LIN {X 0,Y 77.995,Z 481.721,A -85,B 0,C 180,E1 -30607.645,E2 -30607.645} C_VEL
LIN {X 0,Y 72.024,Z 491.434,A -85,B 0,C 180,E1 -30608.921,E2 -30608.921} C_VEL
LIN {X 0,Y 64.422,Z 501.593,A -85,B 0,C 180,E1 -30610.964,E2 -30610.964} C_VEL
LIN {X 0,Y 55.946,Z 510.931,A -85,B 0,C 180,E1 -30613.993,E2 -30613.993} C_VEL
LIN {X 0,Y 48.02,Z 518.337,A -85,B 0,C 180,E1 -30617.976,E2 -30617.976} C_VEL
LIN {X 0,Y 38.72,Z 525.749,A -85,B 0,C 180,E1 -30624.852,E2 -30624.852} C_VEL
LIN {X 0,Y 30.186,Z 531.666,A -85,B 0,C 180,E1 -30635.441,E2 -30635.441} C_VEL
LIN {X 0,Y 23.499,Z 536.326,A -85,B 0,C 180,E1 -30653.279,E2 -30653.279} C_VEL
LIN {X 0,Y 20.813,Z 538.779,A -85,B 0,C 180,E1 -30670.28,E2 -30670.28} C_VEL
LIN {X 0,Y 20.096,Z 540.766,A -85,B 0,C 180,E1 -30690.015,E2 -30690.015} C_VEL
LIN {X 0,Y 20.854,Z 542.293,A -85,B 0,C 180,E1 -30709.71,E2 -30709.71} C_VEL
LIN {X 0,Y 23.631,Z 543.406,A -85,B 0,C 180,E1 -30726.514,E2 -30726.514} C_VEL
LIN {X 0,Y 33.09,Z 544.394,A -85,B 0,C 180,E1 -30748.179,E2 -30748.179} C_VEL
LIN {X 0,Y 45.153,Z 543.887,A -85,B 0,C 180,E1 -30759.066,E2 -30759.066} C_VEL
LIN {X 0,Y 51.564,Z 543.027,A -85,B 0,C 180,E1 -30762.585,E2 -30762.585} C_VEL
LIN {X 0,Y 64.818,Z 540.118,A -85,B 0,C 180,E1 -30767.397,E2 -30767.397} C_VEL
LIN {X 0,Y 74.959,Z 536.824,A -85,B 0,C 180,E1 -30769.904,E2 -30769.904} C_VEL
LIN {X 0,Y 85.212,Z 532.49,A -85,B 0,C 180,E1 -30771.796,E2 -30771.796} C_VEL
LIN {X 0,Y 97.293,Z 525.973,A -85,B 0,C 180,E1 -30773.354,E2 -30773.354} C_VEL
LIN {X 0,Y 107.703,Z 518.838,A -85,B 0,C 180,E1 -30774.356,E2 -30774.356} C_VEL
LIN {X 0,Y 112.916,Z 514.651,A -85,B 0,C 180,E1 -30774.804,E2 -30774.804} C_VEL
LIN {X 0,Y 112.809,Z 514.716,A -85,B 0,C 180,E1 -30775.439,E2 -30775.439} C_VEL
LIN {X 0,Y 101.916,Z 522.899,A -85,B 0,C 180,E1 -30776.583,E2 -30776.583} C_VEL
LIN {X 0,Y 91.427,Z 529.167,A -85,B 0,C 180,E1 -30777.944,E2 -30777.944} C_VEL
LIN {X 0,Y 79.346,Z 534.816,A -85,B 0,C 180,E1 -30780.001,E2 -30780.001} C_VEL
LIN {X 0,Y 70.327,Z 538.074,A -85,B 0,C 180,E1 -30781.999,E2 -30781.999} C_VEL
LIN {X 0,Y 63.406,Z 540.049,A -85,B 0,C 180,E1 -30783.942,E2 -30783.942} C_VEL
LIN {X 0,Y 53.983,Z 542.04,A -85,B 0,C 180,E1 -30787.482,E2 -30787.482} C_VEL
LIN {X 0,Y 43.35,Z 543.328,A -85,B 0,C 180,E1 -30793.385,E2 -30793.385} C_VEL
LIN {X 0,Y 37.114,Z 543.588,A -85,B 0,C 180,E1 -30798.746,E2 -30798.746} C_VEL
LIN {X 0,Y 30.404,Z 543.36,A -85,B 0,C 180,E1 -30807.539,E2 -30807.539} C_VEL
LIN {X 0,Y 22.114,Z 541.861,A -85,B 0,C 180,E1 -30830.518,E2 -30830.518} C_VEL
LIN {X 0,Y 19.731,Z 540.267,A -85,B 0,C 180,E1 -30851.546,E2 -30851.546} C_VEL
LIN {X 0,Y 19.099,Z 538.846,A -85,B 0,C 180,E1 -30868.347,E2 -30868.347} C_VEL
LIN {X 0,Y 19.091,Z 537.172,A -85,B 0,C 180,E1 -30885.573,E2 -30885.573} C_VEL
LIN {X 0,Y 22.808,Z 533.113,A -85,B 0,C 180,E1 -30915.29,E2 -30915.29} C_VEL
LIN {X 0,Y 26.639,Z 530.637,A -85,B 0,C 180,E1 -30924.313,E2 -30924.313} C_VEL
LIN {X 0,Y 28.148,Z 529.719,A -85,B 0,C 180,E1 -30926.304,E2 -30926.304} C_VEL
LIN {X 0,Y 38.83,Z 522.853,A -85,B 0,C 180,E1 -30934.8,E2 -30934.8} C_VEL
LIN {X 0,Y 48.8,Z 515.029,A -85,B 0,C 180,E1 -30939.388,E2 -30939.388} C_VEL
LIN {X 0,Y 57.26,Z 507.041,A -85,B 0,C 180,E1 -30942.012,E2 -30942.012} C_VEL
LIN {X 0,Y 65.835,Z 497.276,A -85,B 0,C 180,E1 -30943.88,E2 -30943.88} C_VEL
LIN {X 0,Y 73.637,Z 486.368,A -85,B 0,C 180,E1 -30945.075,E2 -30945.075} C_VEL
LIN {X 0,Y 79.638,Z 475.755,A -85,B 0,C 180,E1 -30946.09,E2 -30946.09} C_VEL
LIN {X 0,Y 85.204,Z 463.02,A -85,B 0,C 180,E1 -30946.976,E2 -30946.976} C_VEL
LIN {X 0,Y 89.274,Z 450.18,A -85,B 0,C 180,E1 -30947.615,E2 -30947.615} C_VEL
LIN {X 0,Y 91.91,Z 437.116,A -85,B 0,C 180,E1 -30948.013,E2 -30948.013} C_VEL
LIN {X 0,Y 92.458,Z 433.099,A -85,B 0,C 180,E1 -30948.178,E2 -30948.178} C_VEL
LIN {X 0,Y 92.246,Z 431.32,A -85,B 0,C 180,E1 -30951.853,E2 -30951.853} C_VEL
LIN {X 0,Y 92.25,Z 430.805,A -85,B 0,C 180,E1 -30955.63,E2 -30955.63} C_VEL
LIN {X 0,Y 92.334,Z 431.487,A -85,B 0,C 180,E1 -30958.091,E2 -30958.091} C_VEL
LIN {X 0,Y 92.506,Z 433,A -85,B 0,C 180,E1 -30960.668,E2 -30960.668} C_VEL
LIN {X 0,Y 90.295,Z 446.232,A -85,B 0,C 180,E1 -30960.99,E2 -30960.99} C_VEL
LIN {X 0,Y 86.533,Z 459.67,A -85,B 0,C 180,E1 -30961.452,E2 -30961.452} C_VEL
LIN {X 0,Y 82.617,Z 469.744,A -85,B 0,C 180,E1 -30961.86,E2 -30961.86} C_VEL
LIN {X 0,Y 76.497,Z 481.913,A -85,B 0,C 180,E1 -30962.508,E2 -30962.508} C_VEL
LIN {X 0,Y 70.397,Z 491.554,A -85,B 0,C 180,E1 -30963.38,E2 -30963.38} C_VEL
LIN {X 0,Y 63.448,Z 500.632,A -85,B 0,C 180,E1 -30964.576,E2 -30964.576} C_VEL
LIN {X 0,Y 54.828,Z 509.947,A -85,B 0,C 180,E1 -30966.645,E2 -30966.645} C_VEL
LIN {X 0,Y 46.073,Z 517.806,A -85,B 0,C 180,E1 -30969.562,E2 -30969.562} C_VEL
LIN {X 0,Y 36.296,Z 525.123,A -85,B 0,C 180,E1 -30974.534,E2 -30974.534} C_VEL
LIN {X 0,Y 26.69,Z 531.123,A -85,B 0,C 180,E1 -30982.866,E2 -30982.866} C_VEL
LIN {X 0,Y 18.291,Z 535.858,A -85,B 0,C 180,E1 -30999.81,E2 -30999.81} C_VEL
LIN {X 0,Y 13.213,Z 539.446,A -85,B 0,C 180,E1 -31034.6,E2 -31034.6} C_VEL
LIN {X 0,Y 12.988,Z 540.398,A -85,B 0,C 180,E1 -31050.023,E2 -31050.023} C_VEL
LIN {X 0,Y 14.361,Z 541.957,A -85,B 0,C 180,E1 -31079.322,E2 -31079.322} C_VEL
LIN {X 0,Y 18.405,Z 543.114,A -85,B 0,C 180,E1 -31099.814,E2 -31099.814} C_VEL
LIN {X 0,Y 23.846,Z 543.844,A -85,B 0,C 180,E1 -31112.174,E2 -31112.174} C_VEL
LIN {X 0,Y 29.951,Z 544.179,A -85,B 0,C 180,E1 -31119.843,E2 -31119.843} C_VEL
LIN {X 0,Y 43.122,Z 543.735,A -85,B 0,C 180,E1 -31127.955,E2 -31127.955} C_VEL
LIN {X 0,Y 49.9,Z 542.933,A -85,B 0,C 180,E1 -31130.398,E2 -31130.398} C_VEL
LIN {X 0,Y 63.646,Z 540.088,A -85,B 0,C 180,E1 -31133.661,E2 -31133.661} C_VEL
LIN {X 0,Y 70.572,Z 538.062,A -85,B 0,C 180,E1 -31134.821,E2 -31134.821} C_VEL
LIN {X 0,Y 70.453,Z 538.063,A -85,B 0,C 180,E1 -31136.04,E2 -31136.04} C_VEL
LIN {X 0,Y 63.326,Z 540.072,A -85,B 0,C 180,E1 -31137.313,E2 -31137.313} C_VEL
LIN {X 0,Y 52.391,Z 542.311,A -85,B 0,C 180,E1 -31140.001,E2 -31140.001} C_VEL
LIN {X 0,Y 42.26,Z 543.483,A -85,B 0,C 180,E1 -31143.686,E2 -31143.686} C_VEL
LIN {X 0,Y 28.845,Z 543.674,A -85,B 0,C 180,E1 -31152.905,E2 -31152.905} C_VEL
LIN {X 0,Y 22.623,Z 543.135,A -85,B 0,C 180,E1 -31161.222,E2 -31161.222} C_VEL
LIN {X 0,Y 17.145,Z 542.177,A -85,B 0,C 180,E1 -31174.902,E2 -31174.902} C_VEL
LIN {X 0,Y 12.713,Z 540.268,A -85,B 0,C 180,E1 -31207.618,E2 -31207.618} C_VEL
LIN {X 0,Y 15.714,Z 536.78,A -85,B 0,C 180,E1 -31256.546,E2 -31256.546} C_VEL
LIN {X 0,Y 23.204,Z 532.56,A -85,B 0,C 180,E1 -31279.198,E2 -31279.198} C_VEL
LIN {X 0,Y 28.148,Z 529.719,A -85,B 0,C 180,E1 -31286.304,E2 -31286.304} C_VEL
LIN {X 0,Y 32.5,Z 526.943,A -85,B 0,C 180,E1 -31291.777,E2 -31291.777} C_VEL
LIN {X 0,Y 39.201,Z 522.032,A -85,B 0,C 180,E1 -31300.534,E2 -31300.534} C_VEL
LIN {X 0,Y 46.091,Z 516.475,A -85,B 0,C 180,E1 -31306.634,E2 -31306.634} C_VEL
LIN {X 0,Y 50.421,Z 512.681,A -85,B 0,C 180,E1 -31308.273,E2 -31308.273} C_VEL
LIN {X 0,Y 58.971,Z 504.357,A -85,B 0,C 180,E1 -31309.458,E2 -31309.458} C_VEL
LIN {X 0,Y 67.736,Z 493.842,A -85,B 0,C 180,E1 -31310.262,E2 -31310.262} C_VEL
LIN {X 0,Y 74.756,Z 483.422,A -85,B 0,C 180,E1 -31310.772,E2 -31310.772} C_VEL
LIN {X 0,Y 80.851,Z 472.059,A -85,B 0,C 180,E1 -31311.379,E2 -31311.379} C_VEL
LIN {X 0,Y 86.012,Z 459.256,A -85,B 0,C 180,E1 -31311.881,E2 -31311.881} C_VEL
LIN {X 0,Y 89.721,Z 446.196,A -85,B 0,C 180,E1 -31312.28,E2 -31312.28} C_VEL
LIN {X 0,Y 91.253,Z 438.24,A -85,B 0,C 180,E1 -31312.534,E2 -31312.534} C_VEL
LIN {X 0,Y 91.302,Z 437.977,A -85,B 0,C 180,E1 -31316.29,E2 -31316.29} C_VEL
LIN {X 0,Y 88.567,Z 451.042,A -85,B 0,C 180,E1 -31316.585,E2 -31316.585} C_VEL
LIN {X 0,Y 84.456,Z 463.669,A -85,B 0,C 180,E1 -31316.87,E2 -31316.87} C_VEL
LIN {X 0,Y 79.167,Z 475.569,A -85,B 0,C 180,E1 -31317.011,E2 -31317.011} C_VEL
LIN {X 0,Y 72.98,Z 486.443,A -85,B 0,C 180,E1 -31317.485,E2 -31317.485} C_VEL
LIN {X 0,Y 65.927,Z 496.38,A -85,B 0,C 180,E1 -31317.875,E2 -31317.875} C_VEL
LIN {X 0,Y 57.991,Z 505.544,A -85,B 0,C 180,E1 -31318.647,E2 -31318.647} C_VEL
LIN {X 0,Y 48.924,Z 514.175,A -85,B 0,C 180,E1 -31319.998,E2 -31319.998} C_VEL
LIN {X 0,Y 40.425,Z 520.909,A -85,B 0,C 180,E1 -31321.789,E2 -31321.789} C_VEL
LIN {X 0,Y 29.981,Z 527.714,A -85,B 0,C 180,E1 -31325.065,E2 -31325.065} C_VEL
LIN {X 0,Y 18.041,Z 533.94,A -85,B 0,C 180,E1 -31333.189,E2 -31333.189} C_VEL
LIN {X 0,Y 8.82,Z 537.971,A -85,B 0,C 180,E1 -31357.224,E2 -31357.224} C_VEL
LIN {X 0,Y 5.895,Z 540.031,A -85,B 0,C 180,E1 -31410.05,E2 -31410.05} C_VEL
LIN {X 0,Y 8.88,Z 541.621,A -85,B 0,C 180,E1 -31462.374,E2 -31462.374} C_VEL
LIN {X 0,Y 14.843,Z 542.809,A -85,B 0,C 180,E1 -31481.323,E2 -31481.323} C_VEL
LIN {X 0,Y 21.465,Z 543.597,A -85,B 0,C 180,E1 -31489.255,E2 -31489.255} C_VEL
LIN {X 0,Y 28.298,Z 543.965,A -85,B 0,C 180,E1 -31493.518,E2 -31493.518} C_VEL
LIN {X 0,Y 32.634,Z 544.009,A -85,B 0,C 180,E1 -31496.421,E2 -31496.421} C_VEL
LIN {X 0,Y 21.108,Z 543.418,A -85,B 0,C 180,E1 -31502.464,E2 -31502.464} C_VEL
LIN {X 0,Y 14.286,Z 542.495,A -85,B 0,C 180,E1 -31510.193,E2 -31510.193} C_VEL
LIN {X 0,Y 8.122,Z 541.17,A -85,B 0,C 180,E1 -31530.012,E2 -31530.012} C_VEL
LIN {X 0,Y 7.109,Z 538.376,A -85,B 0,C 180,E1 -31619.575,E2 -31619.575} C_VEL
LIN {X 0,Y 12.428,Z 536.133,A -85,B 0,C 180,E1 -31644.264,E2 -31644.264} C_VEL
LIN {X 0,Y 22.659,Z 531.458,A -85,B 0,C 180,E1 -31658.475,E2 -31658.475} C_VEL
LIN {X 0,Y 34.648,Z 524.612,A -85,B 0,C 180,E1 -31664.435,E2 -31664.435} C_VEL
LIN {X 0,Y 45.029,Z 517.193,A -85,B 0,C 180,E1 -31667.252,E2 -31667.252} C_VEL
LIN {X 0,Y 50.421,Z 512.681,A -85,B 0,C 180,E1 -31668.273,E2 -31668.273} C_VEL
LIN {X 0,Y 53.726,Z 514.167,A -85,B 0,C 180,E1 -31668.794,E2 -31668.794} C_VEL
LIN {X 0,Y 53.726,Z 600,A -85,B 0,C 180,E1 -31668.794,E2 -31668.794} C_VEL
LIN {X 0,Y 53.726,Z 600,A -85,B 0,C 180,E1 -31668.794,E2 -31668.794}

QRS_NEXT_CUT()

QRS_NEXT()
QRS_HOME()

END
